PROGRAM UnitTests
VAR
    {attribute 'analysis' := '-33'}
    toWin32ErrorCode_Tests : ToWin32ErrorCode_Tests;
END_VAR

TcUnit.RUN();

END_PROGRAM

(* stored: Version 1.1.0.1, ProductVersion 3.1.4024.11
   POU UnitTests: Id {cc8a0e38-2881-4bc0-a9ad-843c806f9d72}, SpecialFunc None *)
